FUNCTION_BLOCK Invoker
VAR
	_myCommand : ITF_Command;
END_VAR

METHOD ExecuteCommand : BOOL
VAR_INPUT
END_VAR
_myCommand.Execute();
ExecuteCommand := true;
END_METHOD

METHOD SetCommand : BOOL
VAR_INPUT
	MyCommand : ITF_Command;
END_VAR
_myCommand := MyCommand;
SetCommand := true;
END_METHOD

END_FUNCTION_BLOCK

(* stored: Version 1.1.0.1, ProductVersion 3.1.4024.12
   POU Invoker: Id {05faecee-4f77-45b5-8bf8-6e6b526dca0a}, SpecialFunc None
   Method ExecuteCommand: Id {f3c441b2-4514-4069-9c99-bdad23bc48ad}
   Method SetCommand: Id {05ebd954-05db-4e1d-b189-ad09bad64c01} *)
